// TIA Portal V18 export
FUNCTION "AHUProxy" : Void   // FC59010, LAD
{ S7_Optimized_Access := 'TRUE' }
VERSION : 0.1
// stored: AutoNumber false, IsIECCheckEnabled false, SetENOAutomatically false, UDAEnableTagReadback false
   VAR_INPUT
      iUnitID : Int;   // 1=AHUFood, 2=AHUNonFood
      iProxyHeaterID : Int;
      iProxyMixingExtractID : Int;
      iProxyExtractDumperID : Int;
      iProxyReserveID : Int;
   END_VAR
BEGIN

REGION Network 1: Heater Analog
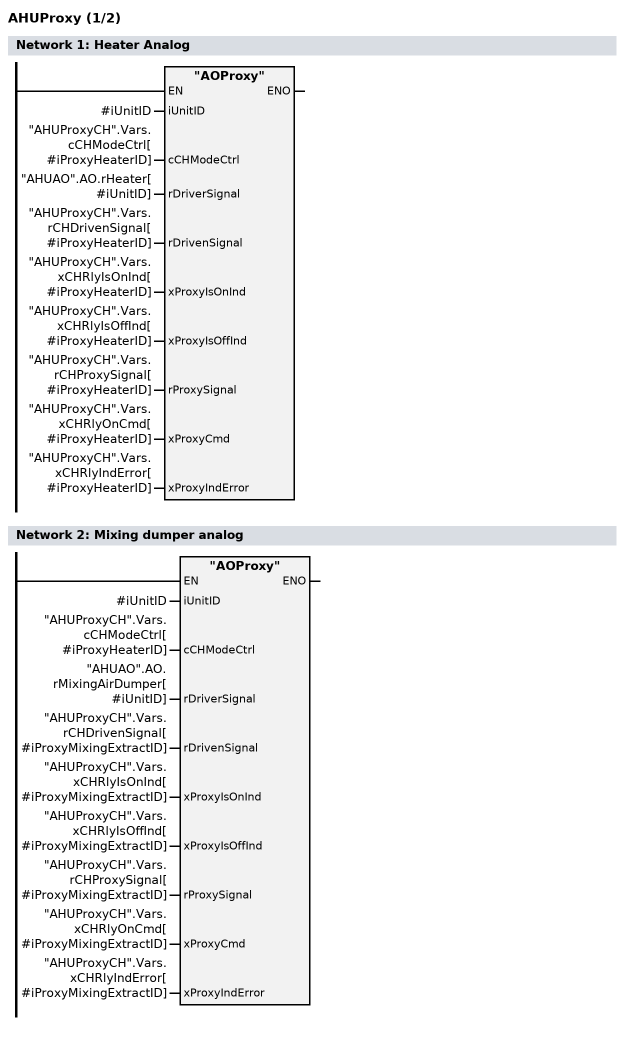
   RUNG wire#powerrail
      "AOProxy"(iUnitID := #iUnitID, cCHModeCtrl := "AHUProxyCH".Vars.cCHModeCtrl[#iProxyHeaterID], rDriverSignal := "AHUAO".AO.rHeater[#iUnitID], rDrivenSignal := "AHUProxyCH".Vars.rCHDrivenSignal[#iProxyHeaterID], xProxyIsOnInd := "AHUProxyCH".Vars.xCHRlyIsOnInd[#iProxyHeaterID], xProxyIsOffInd := "AHUProxyCH".Vars.xCHRlyIsOffInd[#iProxyHeaterID], rProxySignal := "AHUProxyCH".Vars.rCHProxySignal[#iProxyHeaterID], xProxyCmd := "AHUProxyCH".Vars.xCHRlyOnCmd[#iProxyHeaterID], xProxyIndError := "AHUProxyCH".Vars.xCHRlyIndError[#iProxyHeaterID])
   END_RUNG
   // the same network as SCL:
   "AOProxy"(iUnitID := #iUnitID,
             cCHModeCtrl := "AHUProxyCH".Vars.cCHModeCtrl[#iProxyHeaterID],
             rDriverSignal := "AHUAO".AO.rHeater[#iUnitID],
             rDrivenSignal := "AHUProxyCH".Vars.rCHDrivenSignal[#iProxyHeaterID],
             xProxyIsOnInd := "AHUProxyCH".Vars.xCHRlyIsOnInd[#iProxyHeaterID],
             xProxyIsOffInd := "AHUProxyCH".Vars.xCHRlyIsOffInd[#iProxyHeaterID],
             rProxySignal := "AHUProxyCH".Vars.rCHProxySignal[#iProxyHeaterID],
             xProxyCmd := "AHUProxyCH".Vars.xCHRlyOnCmd[#iProxyHeaterID],
             xProxyIndError := "AHUProxyCH".Vars.xCHRlyIndError[#iProxyHeaterID]);
END_REGION

REGION Network 2: Mixing dumper analog
   RUNG wire#powerrail
      "AOProxy"(iUnitID := #iUnitID, cCHModeCtrl := "AHUProxyCH".Vars.cCHModeCtrl[#iProxyHeaterID], rDriverSignal := "AHUAO".AO.rMixingAirDumper[#iUnitID], rDrivenSignal := "AHUProxyCH".Vars.rCHDrivenSignal[#iProxyMixingExtractID], xProxyIsOnInd := "AHUProxyCH".Vars.xCHRlyIsOnInd[#iProxyMixingExtractID], xProxyIsOffInd := "AHUProxyCH".Vars.xCHRlyIsOffInd[#iProxyMixingExtractID], rProxySignal := "AHUProxyCH".Vars.rCHProxySignal[#iProxyMixingExtractID], xProxyCmd := "AHUProxyCH".Vars.xCHRlyOnCmd[#iProxyMixingExtractID], xProxyIndError := "AHUProxyCH".Vars.xCHRlyIndError[#iProxyMixingExtractID])
   END_RUNG
   // the same network as SCL:
   "AOProxy"(iUnitID := #iUnitID,
             cCHModeCtrl := "AHUProxyCH".Vars.cCHModeCtrl[#iProxyHeaterID],
             rDriverSignal := "AHUAO".AO.rMixingAirDumper[#iUnitID],
             rDrivenSignal := "AHUProxyCH".Vars.rCHDrivenSignal[#iProxyMixingExtractID],
             xProxyIsOnInd := "AHUProxyCH".Vars.xCHRlyIsOnInd[#iProxyMixingExtractID],
             xProxyIsOffInd := "AHUProxyCH".Vars.xCHRlyIsOffInd[#iProxyMixingExtractID],
             rProxySignal := "AHUProxyCH".Vars.rCHProxySignal[#iProxyMixingExtractID],
             xProxyCmd := "AHUProxyCH".Vars.xCHRlyOnCmd[#iProxyMixingExtractID],
             xProxyIndError := "AHUProxyCH".Vars.xCHRlyIndError[#iProxyMixingExtractID]);
END_REGION

REGION Network 3: Mixing dumper analog
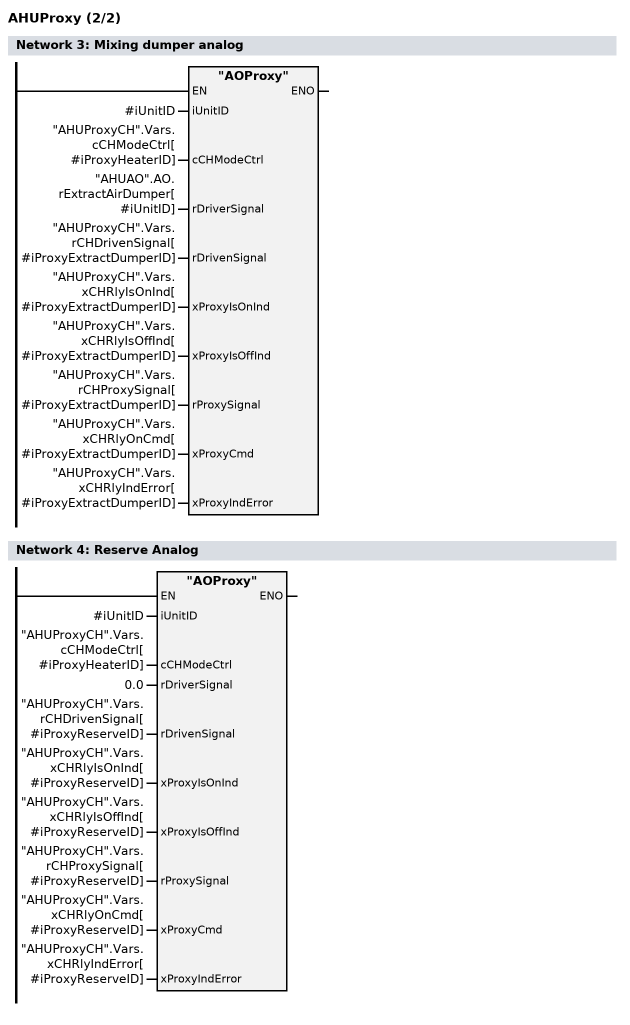
   RUNG wire#powerrail
      "AOProxy"(iUnitID := #iUnitID, cCHModeCtrl := "AHUProxyCH".Vars.cCHModeCtrl[#iProxyHeaterID], rDriverSignal := "AHUAO".AO.rExtractAirDumper[#iUnitID], rDrivenSignal := "AHUProxyCH".Vars.rCHDrivenSignal[#iProxyExtractDumperID], xProxyIsOnInd := "AHUProxyCH".Vars.xCHRlyIsOnInd[#iProxyExtractDumperID], xProxyIsOffInd := "AHUProxyCH".Vars.xCHRlyIsOffInd[#iProxyExtractDumperID], rProxySignal := "AHUProxyCH".Vars.rCHProxySignal[#iProxyExtractDumperID], xProxyCmd := "AHUProxyCH".Vars.xCHRlyOnCmd[#iProxyExtractDumperID], xProxyIndError := "AHUProxyCH".Vars.xCHRlyIndError[#iProxyExtractDumperID])
   END_RUNG
   // the same network as SCL:
   "AOProxy"(iUnitID := #iUnitID,
             cCHModeCtrl := "AHUProxyCH".Vars.cCHModeCtrl[#iProxyHeaterID],
             rDriverSignal := "AHUAO".AO.rExtractAirDumper[#iUnitID],
             rDrivenSignal := "AHUProxyCH".Vars.rCHDrivenSignal[#iProxyExtractDumperID],
             xProxyIsOnInd := "AHUProxyCH".Vars.xCHRlyIsOnInd[#iProxyExtractDumperID],
             xProxyIsOffInd := "AHUProxyCH".Vars.xCHRlyIsOffInd[#iProxyExtractDumperID],
             rProxySignal := "AHUProxyCH".Vars.rCHProxySignal[#iProxyExtractDumperID],
             xProxyCmd := "AHUProxyCH".Vars.xCHRlyOnCmd[#iProxyExtractDumperID],
             xProxyIndError := "AHUProxyCH".Vars.xCHRlyIndError[#iProxyExtractDumperID]);
END_REGION

REGION Network 4: Reserve Analog
   RUNG wire#powerrail
      "AOProxy"(iUnitID := #iUnitID, cCHModeCtrl := "AHUProxyCH".Vars.cCHModeCtrl[#iProxyHeaterID], rDriverSignal := 0.0, rDrivenSignal := "AHUProxyCH".Vars.rCHDrivenSignal[#iProxyReserveID], xProxyIsOnInd := "AHUProxyCH".Vars.xCHRlyIsOnInd[#iProxyReserveID], xProxyIsOffInd := "AHUProxyCH".Vars.xCHRlyIsOffInd[#iProxyReserveID], rProxySignal := "AHUProxyCH".Vars.rCHProxySignal[#iProxyReserveID], xProxyCmd := "AHUProxyCH".Vars.xCHRlyOnCmd[#iProxyReserveID], xProxyIndError := "AHUProxyCH".Vars.xCHRlyIndError[#iProxyReserveID])
   END_RUNG
   // the same network as SCL:
   "AOProxy"(iUnitID := #iUnitID,
             cCHModeCtrl := "AHUProxyCH".Vars.cCHModeCtrl[#iProxyHeaterID],
             rDriverSignal := 0.0,
             rDrivenSignal := "AHUProxyCH".Vars.rCHDrivenSignal[#iProxyReserveID],
             xProxyIsOnInd := "AHUProxyCH".Vars.xCHRlyIsOnInd[#iProxyReserveID],
             xProxyIsOffInd := "AHUProxyCH".Vars.xCHRlyIsOffInd[#iProxyReserveID],
             rProxySignal := "AHUProxyCH".Vars.rCHProxySignal[#iProxyReserveID],
             xProxyCmd := "AHUProxyCH".Vars.xCHRlyOnCmd[#iProxyReserveID],
             xProxyIndError := "AHUProxyCH".Vars.xCHRlyIndError[#iProxyReserveID]);
END_REGION
END_FUNCTION
